{attribute 'qualified_only'}
{attribute 'strict'}
TYPE
    E_ReloadRoundBelt_PickupArea :
    (
        Undefined := 0,
        WareHouseA := 1,
        WareHouseB := 2
        )UINT;
END_TYPE

(* stored: Version 1.1.0.1, ProductVersion 3.1.4024.13
   DUT E_ReloadRoundBelt_PickupArea: Id {cf7e9cb8-d46b-41db-a28f-87954abc5115} *)
